# EPICS substitutions: 300test/evg-fct.subs
file "evg-fct.template"
{
  {
    DEVICE = "fctMap"
  }
}
